{attribute 'no_explicit_call' := 'direct call for this function block is not allowed'}
FUNCTION_BLOCK FB_Recipe IMPLEMENTS  __SYSTEM.IQueryInterface
VAR
	Id 		: T_RecipeId;
	arSteps : ARRAY[0..4] OF T_RecipeStep;
END_VAR

END_FUNCTION_BLOCK

(* stored: Version 1.1.0.1, ProductVersion 3.1.4024.15
   POU FB_Recipe: Id {2c1dce7f-b1a0-4ffd-9ce2-743d05f393b3}, SpecialFunc None *)
